FUNCTION_BLOCK FB_LamparaTemporizada_IL
// La lampara se enciende al accionar el pulsador
// La lampara se apaga transcurrido un tiempo encendidaVAR_INPUT
VAR
    TiempoEncendido   : TIME := T#2S;
END_VAR
VAR_OUTPUT
    TiempoPendiente   : TIME;
END_VAR
VAR
    Temporizador      : TON;
    Lampara   AT %Q*  : BOOL;
    Pulsador  AT %I*  : BOOL;
END_VAR

// NETWORK 1
// instruction list
CAL     Temporizador(
    IN      := Lampara,
    PT      := TiempoEncendido)

// NETWORK 2
// instruction list
LD      TiempoEncendido
SUB     Temporizador.ET
ST      TiempoPendiente

// NETWORK 3
// instruction list
LD      Pulsador
S       Lampara

// NETWORK 4
// instruction list
LD      Temporizador.Q
R       Lampara

END_FUNCTION_BLOCK

(* stored: Version 1.1.0.1, ProductVersion 3.1.4024.15
   POU FB_LamparaTemporizada_IL: Id {40e65883-4b53-4eb1-8d08-bdcbc299153f}, SpecialFunc None *)
